FUNCTION VecNorm : lreal
VAR_INPUT
	a : Vec3;
END_VAR
VAR
END_VAR

VecNorm := SQRT(a.data[0] * a.data[0] + a.data[1] * a.data[1] + a.data[2] * a.data[2]);

END_FUNCTION

(* stored: Version 1.1.0.1, ProductVersion 3.1.4024.2
   POU VecNorm: Id {fa0ebb31-90ed-46d8-88ee-d9f627f7e92a}, SpecialFunc None *)
